Fanuc KAREL source: IO0060.KL

PROGRAM IO0060
%STACKSIZE=65535
%PRIORITY=65535
%NOLOCKGROUP
ROUTINE RTEST FROM IO0060
ROUTINE RTEST
VAR
L1 : ARRAY[3] OF INTEGER
L2 : XYZWPR
L3 : JOINTPOS9
L4 : POSITION
U2C_37 : INTEGER
U2C_38 : REAL
U2C_39 : REAL
U2C_40 : BOOLEAN
U2C_41 : REAL
BEGIN
U2C_37=1
L1[1]=2
U2C_40=TRUE
U2C_41=1.0
-- UNRESOLVED_PC line 19 opcodes [21 21 9D 52 1A] marker_code=77
END RTEST
BEGIN
RTEST
END IO0060
